// TIA Portal V17 export
// export: Created 2023-09-10T16:28:25.2968088Z, ExportSetting WithDefaults, DisplayName Totally Integrated Automation Portal, DisplayVersion V17, DisplayName TIA Portal Openness, DisplayVersion V17, DisplayName TIA Portal Version Control Interface, DisplayVersion V17, DisplayName STEP 7 Professional, DisplayVersion V17, DisplayName STEP 7 Safety, DisplayVersion V17, DisplayName WinCC Advanced, DisplayVersion V17
VAR_GLOBAL   // PLC tag table "Default tag table"
   System_Byte AT %MB1 : Byte;
   FirstScan AT %M1.0 : Bool;
   DiagStatusUpdate AT %M1.1 : Bool;
   AlwaysTRUE AT %M1.2 : Bool;
   AlwaysFALSE AT %M1.3 : Bool;
   Clock_Byte AT %MB0 : Byte;
   Clock_10Hz AT %M0.0 : Bool;
   Clock_5Hz AT %M0.1 : Bool;
   "Clock_2.5Hz" AT %M0.2 : Bool;
   Clock_2Hz AT %M0.3 : Bool;
   "Clock_1.25Hz" AT %M0.4 : Bool;
   Clock_1Hz AT %M0.5 : Bool;
   "Clock_0.625Hz" AT %M0.6 : Bool;
   "Clock_0.5Hz" AT %M0.7 : Bool;
   lastEncoderValue AT %MW8 : Int;
   encoderNumberOfTurn AT %MD10 : DInt;
   machinePosition AT %MD14 : DInt;
   goToPosition AT %M2.0 : Bool;
   broken0 AT %Q0.0 : Bool;
   broken1 AT %Q0.1 : Bool;
   baseSensor AT %I0.0 : Bool;
   stepperMotor_Direction AT %Q0.3 : Bool;
   stepperMotor_Pulse AT %Q0.2 : Bool;
   jogBackward AT %M2.1 : Bool;
   baseReq AT %M2.2 : Bool;
   jogBackwardFromSetpoint AT %M2.3 : Bool;
   jogForward AT %M2.4 : Bool;
   jogForwardFromSetpoint AT %M2.5 : Bool;
   memoryBit0 AT %M2.6 : Bool;
   memoryBit1 AT %M2.7 : Bool;
   inPosition AT %M3.0 : Bool;
   memoryBit2 AT %M3.1 : Bool;
   memoryBit3 AT %M3.2 : Bool;
   homing AT %M3.3 : Bool;
   homingDone AT %M3.4 : Bool;
   memoryBit4 AT %M3.5 : Bool;
   memoryBit5 AT %M3.6 : Bool;
   homingStep1 AT %M3.7 : Bool;
   homingStep2 AT %M4.0 : Bool;
   memoryBit6 AT %M4.1 : Bool;
   homingStep3 AT %M4.2 : Bool;
   memoryBit7 AT %M4.3 : Bool;
   seqNum AT %MW6 : Int;
   memoryBit8 AT %M4.4 : Bool;
   memoryBit9 AT %M4.5 : Bool;
   memoryBit10 AT %M4.6 : Bool;
   checkPositionAfterReboot AT %M4.7 : Bool;
   memoryBit11 AT %M5.0 : Bool;
   positionNotActual AT %M5.1 : Bool;
END_VAR
